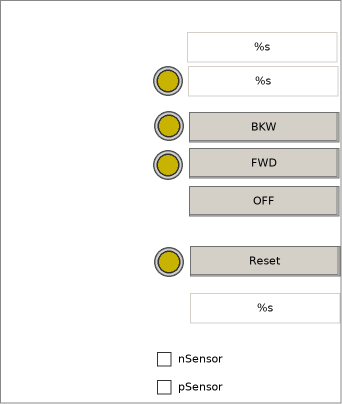
VISUALIZATION V_piston  // 342x404
VAR_IN_OUT
	p : piston;
END_VAR
    Textfield (187,32 150x30), "%s", text variable: p.pistonName
    Button (189,148 150x30), "FWD"
        OnMouseClick: execute { P.fwd(); }
    Textfield (188,66 150x30), "%s", text variable: p.sState
    Button (189,112 150x30), "BKW"
        OnMouseClick: execute { P.bkw(); }
    Button (189,186 150x30), "OFF"
        OnMouseClick: execute { P.off(); }
    Button (190,246 150x30), "Reset"
        OnMouseClick: execute { P.reset(); }
    Lamp1 (152,245 34x34), variable: p.error, style: Lamp-Lamp1-Yellow
    Lamp1 (151,64 34x34), variable: p.busy, style: Lamp-Lamp1-Yellow
    Textfield (190,293 150x30), "%s", text variable: p.errormessage
    Checkbox (155,344 150x30), "nSensor", variable: p.nSensor
    Checkbox (155,372 150x30), "pSensor", variable: p.pSensor
    Lamp1 (152,109 34x34), variable: p.nOut, style: Lamp-Lamp1-Yellow
    Lamp1 (151,148 34x34), variable: p.pOut, style: Lamp-Lamp1-Yellow
END_VISUALIZATION

(* stored: Version 1.1.0.1, ProductVersion 3.1.4022.18
   Visu V_piston: Id {8f943f64-6b64-4da3-9ebc-bb30c1203a19} *)
